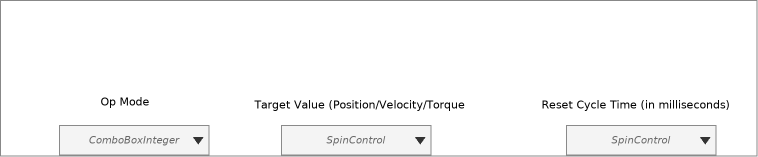
VISUALIZATION Visualization  // 758x157
    ComboBoxInteger (59,125 150x30), variable: GVL.opmode, text list: 'OpMode'
    SpinControl (281,125 150x30), variable: GVL.TARGET_AMPLITUDE
    Label (50,87 150x30), "Op Mode"
    Label (241,89 238x32), "Target Value (Position/Velocity/Torque"
    SpinControl (566,125 150x30), variable: GVL.RESET_SIGNAL
    Label (516,90 240x30), "Reset Cycle Time (in milliseconds)"
END_VISUALIZATION

(* stored: Version 1.1.0.1, ProductVersion 3.1.4022.16
   Visu Visualization: Id {813f488e-bff5-490a-b1e4-0c06e4dbaec8} *)
